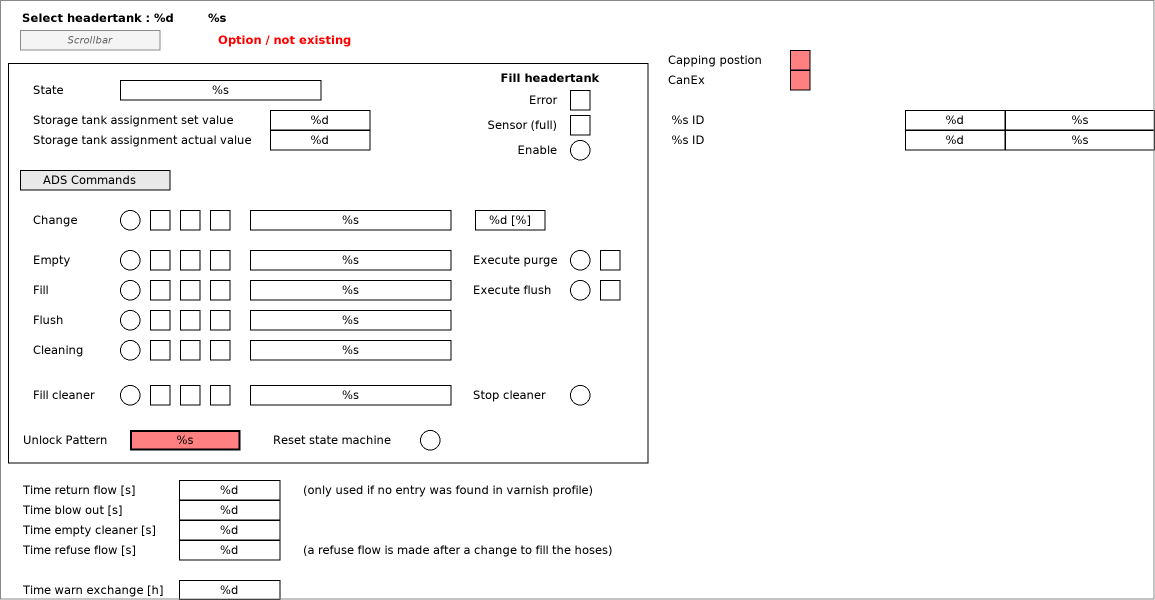
VISUALIZATION VISU_HEADERTANK  // 1155x600
    Rectangle (8,63 640x400)
    Rectangle (30,310 80x20), "Flush"
    Ellipse (120,310 20x20), colour toggle: PRG_INK.sAdsIkHeaderTank[PRG_INK.iL_Sel_HeaderTank].sI_CommandFlush.bI_Command, input disabled if: NOT PRG_INK.sAdsIkHeaderTank[PRG_INK.iL_Sel_HeaderTank].sI_CommandFlush.bO_CommandCanEx
        tap PRG_INK.sAdsIkHeaderTank[PRG_INK.iL_Sel_HeaderTank].sI_CommandFlush.bI_Command
    Rectangle (20,170 150x20)
    Rectangle (40,170 130x20), "ADS Commands"
    RoundedRectangle (150,310 20x20), tooltip "CanEx", colour toggle: PRG_INK.sAdsIkHeaderTank[PRG_INK.iL_Sel_HeaderTank].sI_CommandFlush.bO_CommandCanEx
    RoundedRectangle (210,310 20x20), tooltip "Exec", colour toggle: PRG_INK.sAdsIkHeaderTank[PRG_INK.iL_Sel_HeaderTank].sI_CommandFlush.bO_CommandExec
    RoundedRectangle (180,310 20x20), tooltip "CanStop", colour toggle: PRG_INK.sAdsIkHeaderTank[PRG_INK.iL_Sel_HeaderTank].sI_CommandFlush.bO_CommandCanStop
    Scrollbar (20,30 140x20), tooltip "y-shift"
        p2245068023: CONFIGURATION.iCIk_NB_HEADERTANK
        p1057716461: PRG_INK.iL_Sel_HeaderTank
    Rectangle (15,8 180x20), "Select headertank : %d", text variable: PRG_INK.iL_Sel_HeaderTank
    Rectangle (30,340 80x20), "Cleaning"
    Ellipse (120,340 20x20), colour toggle: PRG_INK.sAdsIkHeaderTank[PRG_INK.iL_Sel_HeaderTank].sI_CommandCleaning.bI_Command, input disabled if: NOT PRG_INK.sAdsIkHeaderTank[PRG_INK.iL_Sel_HeaderTank].sI_CommandCleaning.bO_CommandCanEx
        tap PRG_INK.sAdsIkHeaderTank[PRG_INK.iL_Sel_HeaderTank].sI_CommandCleaning.bI_Command
    RoundedRectangle (150,340 20x20), tooltip "CanEx", colour toggle: PRG_INK.sAdsIkHeaderTank[PRG_INK.iL_Sel_HeaderTank].sI_CommandCleaning.bO_CommandCanEx
    RoundedRectangle (210,340 20x20), tooltip "Exec", colour toggle: PRG_INK.sAdsIkHeaderTank[PRG_INK.iL_Sel_HeaderTank].sI_CommandCleaning.bO_CommandExec
    RoundedRectangle (180,340 20x20), tooltip "CanStop", colour toggle: PRG_INK.sAdsIkHeaderTank[PRG_INK.iL_Sel_HeaderTank].sI_CommandCleaning.bO_CommandCanStop
    Rectangle (30,280 80x20), "Fill"
    Ellipse (120,280 20x20), colour toggle: PRG_INK.sAdsIkHeaderTank[PRG_INK.iL_Sel_HeaderTank].sI_CommandFill.bI_Command, input disabled if: NOT PRG_INK.sAdsIkHeaderTank[PRG_INK.iL_Sel_HeaderTank].sI_CommandFill.bO_CommandCanEx
        tap PRG_INK.sAdsIkHeaderTank[PRG_INK.iL_Sel_HeaderTank].sI_CommandFill.bI_Command
    RoundedRectangle (150,280 20x20), tooltip "CanEx", colour toggle: PRG_INK.sAdsIkHeaderTank[PRG_INK.iL_Sel_HeaderTank].sI_CommandFill.bO_CommandCanEx
    RoundedRectangle (210,280 20x20), tooltip "Exec", colour toggle: PRG_INK.sAdsIkHeaderTank[PRG_INK.iL_Sel_HeaderTank].sI_CommandFill.bO_CommandExec
    RoundedRectangle (180,280 20x20), tooltip "CanStop", colour toggle: PRG_INK.sAdsIkHeaderTank[PRG_INK.iL_Sel_HeaderTank].sI_CommandFill.bO_CommandCanStop
    Rectangle (30,250 80x20), "Empty"
    Ellipse (120,250 20x20), colour toggle: PRG_INK.sAdsIkHeaderTank[PRG_INK.iL_Sel_HeaderTank].sI_CommandEmpty.bI_Command, input disabled if: NOT PRG_INK.sAdsIkHeaderTank[PRG_INK.iL_Sel_HeaderTank].sI_CommandEmpty.bO_CommandCanEx
        tap PRG_INK.sAdsIkHeaderTank[PRG_INK.iL_Sel_HeaderTank].sI_CommandEmpty.bI_Command
    RoundedRectangle (150,250 20x20), tooltip "CanEx", colour toggle: PRG_INK.sAdsIkHeaderTank[PRG_INK.iL_Sel_HeaderTank].sI_CommandEmpty.bO_CommandCanEx
    RoundedRectangle (210,250 20x20), tooltip "Exec", colour toggle: PRG_INK.sAdsIkHeaderTank[PRG_INK.iL_Sel_HeaderTank].sI_CommandEmpty.bO_CommandExec
    RoundedRectangle (180,250 20x20), tooltip "CanStop", colour toggle: PRG_INK.sAdsIkHeaderTank[PRG_INK.iL_Sel_HeaderTank].sI_CommandEmpty.bO_CommandCanStop
    Rectangle (250,250 201x20), "%s", text variable: PRG_INK.fb_Headertank[PRG_INK.iL_Sel_HeaderTank].aL_StateEmpty
    Rectangle (250,280 201x20), "%s", text variable: PRG_INK.fb_Headertank[PRG_INK.iL_Sel_HeaderTank].aL_StateFill
    Rectangle (250,310 201x20), "%s", text variable: PRG_INK.fb_Headertank[PRG_INK.iL_Sel_HeaderTank].aL_StateFlush
    Rectangle (250,340 201x20), "%s", text variable: PRG_INK.fb_Headertank[PRG_INK.iL_Sel_HeaderTank].aL_StateCleaning
    Rectangle (470,280 90x20), "Execute flush"
    Ellipse (570,280 20x20), colour toggle: PRG_INK.fb_Headertank[PRG_INK.iL_Sel_HeaderTank].bL_ExecuteFlushManu
        toggle PRG_INK.fb_Headertank[PRG_INK.iL_Sel_HeaderTank].bL_ExecuteFlushManu
    Rectangle (30,210 80x20), "Change"
    Ellipse (120,210 20x20), colour toggle: PRG_INK.sAdsIkHeaderTank[PRG_INK.iL_Sel_HeaderTank].sI_CommandChange.bI_Command, input disabled if: NOT PRG_INK.sAdsIkHeaderTank[PRG_INK.iL_Sel_HeaderTank].sI_CommandChange.bO_CommandCanEx
        tap PRG_INK.sAdsIkHeaderTank[PRG_INK.iL_Sel_HeaderTank].sI_CommandChange.bI_Command
    RoundedRectangle (150,210 20x20), tooltip "CanEx", colour toggle: PRG_INK.sAdsIkHeaderTank[PRG_INK.iL_Sel_HeaderTank].sI_CommandChange.bO_CommandCanEx
    RoundedRectangle (210,210 20x20), tooltip "Exec", colour toggle: PRG_INK.sAdsIkHeaderTank[PRG_INK.iL_Sel_HeaderTank].sI_CommandChange.bO_CommandExec
    RoundedRectangle (180,210 20x20), tooltip "CanStop", colour toggle: PRG_INK.sAdsIkHeaderTank[PRG_INK.iL_Sel_HeaderTank].sI_CommandChange.bO_CommandCanStop
    Rectangle (250,210 201x20), "%s", text variable: PRG_INK.fb_Headertank[PRG_INK.iL_Sel_HeaderTank].aL_StateChange
    Rectangle (270,110 100x20), "%d", text variable: PRG_INK.sAdsIkHeaderTank[PRG_INK.iL_Sel_HeaderTank].sI_StoragetankAssignment.lI_Val
        OnMouseDown: write the text variable via Default
    Rectangle (30,110 230x20), "Storage tank assignment set value"
    Rectangle (270,130 100x20), "%d", text variable: PRG_INK.sAdsIkHeaderTank[PRG_INK.iL_Sel_HeaderTank].sO_ActStoragetankAssignment.lI_Val
        OnMouseDown: write the text variable via Edit
    Rectangle (30,130 230x20), "Storage tank assignment actual value"
    RoundedRectangle (600,280 20x20), colour toggle: PRG_INK.fb_Headertank[PRG_INK.iL_Sel_HeaderTank].bL_ExecuteFlush
    Rectangle (120,80 201x20), "%s", text variable: PRG_INK.fb_Headertank[PRG_INK.iL_Sel_HeaderTank].eL_StateHeadertank
    Rectangle (179,480 101x20), "%d", text variable: PRG_INK.lL_TimeReturnFlow
        OnMouseDown: write the text variable via Edit
    Rectangle (20,480 147x20), "Time return flow [s]"
    Rectangle (179,500 101x20), "%d", text variable: PRG_INK.lL_TimeBlowOut
        OnMouseDown: write the text variable via Edit
    Rectangle (20,500 147x20), "Time blow out [s]"
    Rectangle (179,520 101x20), "%d", text variable: PRG_INK.lL_TimeEmptyCleaner
        OnMouseDown: write the text variable via Edit
    Rectangle (20,520 147x20), "Time empty cleaner [s]"
    Rectangle (179,580 101x20), "%d", text variable: PRG_INK.lL_TimeWarnExchange
        OnMouseDown: write the text variable via Edit
    Rectangle (20,580 147x20), "Time warn exchange [h]"
    Rectangle (470,90 90x20), "Error"
    RoundedRectangle (570,90 20x20), colour toggle: PRG_INK.sAdsIkHeaderTank[PRG_INK.iL_Sel_HeaderTank].sI_AckFillInk.bO_CommandCanEx
    Rectangle (30,80 80x20), "State"
    Ellipse (570,140 20x20), colour toggle: PRG_INK.sAdsIkHeaderTank[PRG_INK.iL_Sel_HeaderTank].bI_EnableFillInk
        toggle PRG_INK.sAdsIkHeaderTank[PRG_INK.iL_Sel_HeaderTank].bI_EnableFillInk
    Rectangle (470,140 90x20), "Enable"
    Rectangle (470,115 90x20), "Sensor (full)"
    RoundedRectangle (570,115 20x20), colour toggle: (PRG_INK.sAdsIkHeaderTank[PRG_INK.iL_Sel_HeaderTank].cO_StatusFillInk.5) <> 0
    Rectangle (20,430 100x20), "Unlock Pattern"
    Rectangle (130,430 110x20), "%s", text variable: PRG_INK.fb_Headertank[PRG_INK.iL_Sel_HeaderTank].aI_SafePattern, colour toggle: PRG_INK.fb_Headertank[PRG_INK.iL_Sel_HeaderTank].bL_Unlock
        OnMouseDown: write the text variable via Edit
    Ellipse (420,430 20x20), colour toggle: PRG_INK.fb_Headertank[PRG_INK.iL_Sel_HeaderTank].fb_RTrigStateMachineReset.CLK, invisible if: NOT PRG_INK.fb_Headertank[PRG_INK.iL_Sel_HeaderTank].bL_Unlock
        tap PRG_INK.fb_Headertank[PRG_INK.iL_Sel_HeaderTank].fb_RTrigStateMachineReset.CLK
    Rectangle (270,430 140x20), "Reset state machine", invisible if: NOT PRG_INK.fb_Headertank[PRG_INK.iL_Sel_HeaderTank].bL_Unlock
    Rectangle (905,110 100x20), "%d", text variable: PRG_INK.sL_BLK_INKSTORAGE_TANK[1].iBlk_AdsId
        OnMouseDown: write the text variable via Edit
    Rectangle (665,110 230x20), "%s ID", text variable: PRG_INK.sAdsIkInkStorageTank[1].aO_Name
    RoundedRectangle (790,70 20x20), colour toggle: PRG_INK.bL_HeadertankCanEx
        toggle PRG_INK.sAdsIkHeaderTank[PRG_INK.iL_Sel_HeaderTank].bI_EnableFillInk
    Rectangle (665,70 110x20), "CanEx"
    Rectangle (300,480 300x20), "(only used if no entry was found in varnish profile)"
    Rectangle (475,210 70x20), "%d [%]", text variable: PRG_INK.fb_Headertank[PRG_INK.iL_Sel_HeaderTank].iL_PercentStateChange
        OnMouseDown: write the text variable via Edit
    Rectangle (495,68 110x20), "Fill headertank"
    Rectangle (30,385 80x20), "Fill cleaner"
    Ellipse (120,385 20x20), colour toggle: PRG_INK.sAdsIkHeaderTank[PRG_INK.iL_Sel_HeaderTank].sI_ActivateCleaner.bI_Command, input disabled if: NOT PRG_INK.sAdsIkHeaderTank[PRG_INK.iL_Sel_HeaderTank].sI_ActivateCleaner.bO_CommandCanEx
        tap PRG_INK.sAdsIkHeaderTank[PRG_INK.iL_Sel_HeaderTank].sI_ActivateCleaner.bI_Command
    RoundedRectangle (150,385 20x20), tooltip "CanEx", colour toggle: PRG_INK.sAdsIkHeaderTank[PRG_INK.iL_Sel_HeaderTank].sI_ActivateCleaner.bO_CommandCanEx
    RoundedRectangle (210,385 20x20), tooltip "Exec", colour toggle: PRG_INK.sAdsIkHeaderTank[PRG_INK.iL_Sel_HeaderTank].sI_ActivateCleaner.bO_CommandExec
    RoundedRectangle (180,385 20x20), tooltip "CanStop", colour toggle: PRG_INK.sAdsIkHeaderTank[PRG_INK.iL_Sel_HeaderTank].sI_ActivateCleaner.bO_CommandCanStop
    Rectangle (250,385 201x20), "%s", text variable: PRG_INK.fb_Headertank[PRG_INK.iL_Sel_HeaderTank].aL_StateCleaner
    RoundedRectangle (790,50 20x20), colour toggle: PRG_INK.iMachineInk[iCIk_MAP_HEADERTANK_HT_GROUP[PRG_INK.iL_Sel_HeaderTank]].pInCappingPos
        toggle PRG_INK.sAdsIkHeaderTank[PRG_INK.iL_Sel_HeaderTank].bI_EnableFillInk
    Rectangle (665,50 110x20), "Capping postion"
    Rectangle (215,30 150x20), "Option / not existing", invisible if: bCIk_HEADERTANK_EXIST[PRG_INK.iL_Sel_HeaderTank]
    Rectangle (470,385 90x20), "Stop cleaner"
    Ellipse (570,385 20x20), colour toggle: PRG_INK.bIDp_StopFillCleaner[PRG_INK.iL_Sel_HeaderTank]
        tap PRG_INK.bIDp_StopFillCleaner[PRG_INK.iL_Sel_HeaderTank]
    Rectangle (905,130 100x20), "%d", text variable: PRG_INK.sL_BLK_INKSTORAGE_TANK[2].iBlk_AdsId
        OnMouseDown: write the text variable via Edit
    Rectangle (665,130 230x20), "%s ID", text variable: PRG_INK.sAdsIkInkStorageTank[2].aO_Name
    Rectangle (205,8 180x20), "%s", text variable: PRG_INK.sC_Config_I.aC_HEADERTANKGROUP_NAME_DETAIL[iCIk_MAP_HEADERTANK_HT_GROUP[PRG_INK.iL_Sel_HeaderTank]]
    Rectangle (1005,110 150x20), "%s", text variable: PRG_INK.sAdsIkInkStorageTank[1].sI_InkParameter.aColorName
        OnMouseDown: write the text variable via Edit
    Rectangle (1005,130 150x20), "%s", text variable: PRG_INK.sAdsIkInkStorageTank[2].sI_InkParameter.aColorName
        OnMouseDown: write the text variable via Edit
    Rectangle (179,540 101x20), "%d", text variable: PRG_INK.lL_TimeRefuseFlow
        OnMouseDown: write the text variable via Edit
    Rectangle (20,540 147x20), "Time refuse flow [s]"
    Rectangle (300,540 344x20), "(a refuse flow is made after a change to fill the hoses)"
    Rectangle (470,250 96x20), "Execute purge"
    Ellipse (570,250 20x20), colour toggle: PRG_INK.fb_Headertank[PRG_INK.iL_Sel_HeaderTank].bI_ExecutePurgeManu
        toggle PRG_INK.fb_Headertank[PRG_INK.iL_Sel_HeaderTank].bI_ExecutePurgeManu
    RoundedRectangle (600,250 20x20), colour toggle: PRG_INK.fb_Headertank[PRG_INK.iL_Sel_HeaderTank].bL_SkipPurge
END_VISUALIZATION

(* stored: Version 1.1.0.1, ProductVersion 3.1.4024.9
   Visu VISU_HEADERTANK: Id {bbd48626-4429-4c1a-ae06-3a5ccdcd2dd3} *)
